// TIA Portal V19 export
TYPE "LUC_typeModes"
// stored: Access Published
   STRUCT
      current : DInt;   // Current operating mode
      production : Bool;   // The operating mode "Production" is active
      maintenance : Bool;   // The operating mode "Maintenance" is active
      manual : Bool;   // The operating mode "Manual" is active
      userMode01 : Bool;   // The operating mode "UserMode1" is active
      userMode02 : Bool;   // The operating mode "UserMode2" is active
      userMode03 : Bool;   // The operating mode "UserMode3" is active
      userMode04 : Bool;   // The operating mode "UserMode4" is active
      userMode05 : Bool;   // The operating mode "UserMode5" is active
      userMode06 : Bool;   // The operating mode "UserMode6" is active
      userMode07 : Bool;   // The operating mode "UserMode7" is active
      userMode08 : Bool;   // The operating mode "UserMode8" is active
      userMode09 : Bool;   // The operating mode "UserMode9" is active
      userMode10 : Bool;   // The operating mode "UserMode10" is active
      userMode11 : Bool;   // The operating mode "UserMode11" is active
      userMode12 : Bool;   // The operating mode "UserMode12" is active
      userMode13 : Bool;   // The operating mode "UserMode13" is active
   END_STRUCT;
END_TYPE
